Staubli VAL3: duplicate.pgx

public program duplicate(string x_sCopy, string x_sPaste, num& x_nResult[])
  local num i
  local num l_nSize
  local string l_sItem
  local bool l_bFound
  local num l_nResult
begin

end
